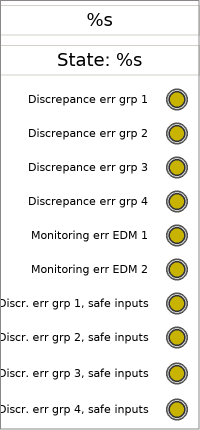
VISUALIZATION DiagEStop  // 200x430
VAR_INPUT
	state:STRING(15);
	bits:st_diagFBBits;
	blockName:STRING(15);
END_VAR
    Label (1,87 150x25), "Discrepance err grp 1"
    Label (1,121 150x25), "Discrepance err grp 2"
    Label (1,155 150x25), "Discrepance err grp 3"
    Label (1,189 150x25), "Discrepance err grp 4"
    Label (1,223 150x25), "Monitoring err EDM 1"
    Label (1,257 150x25), "Monitoring err EDM 2"
    Label (1,291 150x25), "Discr. err grp 1, safe inputs"
    Label (1,325 150x25), "Discr. err grp 2, safe inputs"
    Lamp1 (162,87 30x25), variable: bits[0], style: Lamp-Lamp1-Yellow
    Lamp1 (162,121 30x25), variable: bits[1], style: Lamp-Lamp1-Yellow
    Lamp1 (162,189 30x25), variable: bits[3], style: Lamp-Lamp1-Yellow
    Lamp1 (162,223 30x25), variable: bits[4], style: Lamp-Lamp1-Yellow
    Lamp1 (162,257 30x25), variable: bits[5], style: Lamp-Lamp1-Yellow
    Lamp1 (162,291 30x25), variable: bits[8], style: Lamp-Lamp1-Yellow
    Lamp1 (162,325 30x25), variable: bits[9], style: Lamp-Lamp1-Yellow
    Lamp1 (162,155 30x25), variable: bits[2], style: Lamp-Lamp1-Yellow
    Label (1,361 150x25), "Discr. err grp 3, safe inputs"
    Lamp1 (162,361 30x25), variable: bits[10], style: Lamp-Lamp1-Yellow
    Label (1,397 150x25), "Discr. err grp 4, safe inputs"
    Lamp1 (162,397 30x25), variable: bits[11], style: Lamp-Lamp1-Yellow
    Textfield (0,45 200x30), "State: %s", text variable: state
    Textfield (0,5 200x30), "%s", text variable: blockName
END_VISUALIZATION

(* stored: Version 1.1.0.1, ProductVersion 3.1.4024.12
   Visu DiagEStop: Id {e13d0412-b864-4a3b-b3c2-d055cd820ed8} *)
